(* IEC 61131-3 sources: programs/VI-54/VI-54_20171205/VI-54_20171205/Stations/Screen/LseClass170718/Class/AccessControlUSBDetection, 1 file *)

(* ---- AccessControlUSBDetection.st ---- *)
//"no usb stick is found" value

#define NO_USB 16#FFFF

(*!
<Class
	Name               = "AccessControlUSBDetection"
	Revision           = "1.1"
	RealtimeTask       = "false"
	CyclicTask         = "false"
	BackgroundTask     = "false"
	Sigmatek           = "false"
	OSInterface        = "false"
	HighPriority       = "false"
	Automatic          = "false"
	UpdateMode         = "Prescan"
	SharedCommandTable = "true"
	Objectsize         = "(570,240)"
	Comment            = "This class detects USB-activity.&#13;&#10;Override global-methods USBDeviceIN and USBDeviceOUT for user-defined action on usb-event&#13;&#10;">
	<Channels>
		<Client Name="cFileSys" Required="false" Internal="false" Comment="object channel to FileOp (don&apos;t connect!)"/>
		<Client Name="coAccessControl" Required="true" Internal="false" Comment="object channel - Connect to AccessControlMain object"/>
	</Channels>
	<RevDoku>
		<Owner Company="Sigmatek"/>
		<Dokumentation Revision="1.1" Date="2015-09-22" Company="Sigmatek" Description="Creation."/>
	</RevDoku>
	<Network Name="AccessControlUSBDetection">
		<!-- List of Components in this network -->
		<Components>
			<Object
				Name       = "_base"
				Class      = "_Global"
				Position   = "(218,120)"
				Visualized = "false">
				<Channels>
					<Server Name="Server0"/>
					<Client Name="Lse"/>
				</Channels>
			</Object>
		</Components>
		<Comments>
		</Comments>
		<!-- List of Connections in this network -->
		<Connections>
			<Connection Source="this.Server0" Destination="_base.Server0" Vertices="(690,210),(518,210),"/>
			<Connection Source="_base.Lse" Destination="this.Lse" Vertices="(218,210),(38,210),"/>
		</Connections>
		<!-- Headerfiles -->
		<Options>
		</Options>
	</Network>
</Class>
*)
#pragma using _Global

AccessControlUSBDetection : CLASS
: _Global
	TYPE
	  Letters :
	  (
	    _A,
	    _B,
	    _C,
	    _D,
	    _E,
	    _F,
	    _G,
	    _H,
	    _I,
	    _J,
	    _K,
	    _L,
	    _M,
	    _N,
	    _O,
	    _P,
	    _Q,
	    _R,
	    _S,
	    _T,
	    _U,
	    _V,
	    _W,
	    _X,
	    _Y,
	    _Z
	  )$UDINT;
	  T_SerNum : ARRAY [0..20] OF CHAR;
	END_TYPE
  //Servers:
  //Clients:
	cFileSys 	: CltChCmd__FileSys;
	coAccessControl 	: CltChCmd_AccessControlMain;
  //Variables:
		DriveList : ARRAY [0..25] OF CHAR;

		OldDriveList : ARRAY [0..25] OF CHAR;

		SerNumArray : ARRAY [0..25] OF T_SerNum;

  //Functions:

	FUNCTION VIRTUAL GLOBAL Init;

	FUNCTION VIRTUAL GLOBAL IF_WindowRun
		VAR_INPUT
			whoami 	: ^_WHOAMI;
			pic 	: ^void;
			event 	: ^_EVENT;
		END_VAR;
				//! <Function Comment="Will be called when a usb-stick is plugged in or out. It checks if a serial number of the usb-stick is available." Name="CheckSerNum"/>
	FUNCTION CheckSerNum
		VAR_INPUT
			INorOUT 	: DINT;			//! <Variable Comment="1..usb-stick is plugged in&#13;&#10;2..usb-stick is plugged out" Name="CheckSerNum.INorOUT"/>
		END_VAR;
				//! <Function Comment="Will be called when a usb-stick is plugged in." Name="USBDeviceIN"/>
	FUNCTION VIRTUAL GLOBAL USBDeviceIN
		VAR_INPUT
			pSerNum 	: ^void;			//! <Variable Comment="Pointer to the serial number of the usb-stick." Name="USBDeviceIN.pSerNum"/>
		END_VAR;
				//! <Function Comment="Will be called if a plugged in usb-stick is unplugged." Name="USBDeviceOUT"/>
	FUNCTION VIRTUAL GLOBAL USBDeviceOUT
		VAR_INPUT
			pSerNum 	: ^void;			//! <Variable Comment="Pointer to the serial number of the usb-stick." Name="USBDeviceOUT.pSerNum"/>
		END_VAR;
  //Tables:
	FUNCTION @STD
		VAR_OUTPUT
			ret_code	: CONFSTATES;
		END_VAR;
	FUNCTION GLOBAL TAB @CT_;
END_CLASS;

#pragma usingLtd _FileSys
#pragma usingLtd AccessControlMain

#include " lsl_st_syssernum.h"

FUNCTION VIRTUAL GLOBAL AccessControlUSBDetection::IF_WindowRun
	VAR_INPUT
		whoami 	: ^_WHOAMI;
		pic 	: ^void;
		event 	: ^_EVENT;
	END_VAR

  //call method from baseclass
  _Global::IF_WindowRun(whoami, pic, event);

  if event^.ftype <> _EVENT_NONE then
    //Check if there is some action on the usb-port
    if ( event^.ftype = _EVENT_LASALOS ) & ( event^.scancode = 8 )then

      //Check if usb stick was pluged or draged
      if event^.modifier = 1 | event^.modifier = 2 then

        cFileSys.GetDriveListShort(drivelist:= #DriveList$CHAR); //Get DriveList

        CheckSerNum(INorOUT:=event^.modifier); //check which device was plugged | unplugged

      end_if;
    end_if;
  end_if;

END_FUNCTION

FUNCTION VIRTUAL GLOBAL AccessControlUSBDetection::Init

  //call method from base class
  _Global::init();

  if _firstscan then
   _memset(#OldDriveList, 0, sizeof(OldDriveList));

  end_if;

END_FUNCTION

FUNCTION AccessControlUSBDetection::CheckSerNum
	VAR_INPUT
		INorOUT 	: DINT;
	END_VAR
  VAR
    counter : DINT;
    PISysSernum : ^LSL_ISYSSERNUM;
    Drive : USINT;
    pChar   : ^CHAR;
    retcode : DINT;
    Found : BOOL;
  END_VAR

  //search for all changed USb drives
  for counter := 0 to 25 do

    //if the drive is a UsbDevice, the device has changed since last UsbEvent and the device is plugged in
    if DriveList[counter] = 16#0B & DriveList[counter] <> OldDriveList[counter] & INorOUT = 1 then

      //check if serial number available and not zero
      if OS_CILGET("ISYSSERNUM", #pISysSernum) then
      else

         Drive := 'a' + to_usint(counter);
         _memset(#SerNumArray[counter], 0, sizeof(T_SerNum));
         retcode := ISYSSERNUM_SERNUMGETPLCDRIVE( Drive, #SerNumArray[counter], 20 );
         pChar := #SerNumArray[counter][0];
         Found := FALSE;
         while pChar^ <> 0 do
           if (pChar^ = ' ') | (pChar^ = '0') then
             pChar += sizeof(CHAR);
           else
             Found := TRUE;
             exit;
           end_if;
         end_while;
      end_if;

      if Found then

        USBDeviceIN(#SerNumArray[counter][0]); //call the user definable IN-Method

      end_if;

    //...if the device is unplugged
    elsif OldDriveList[counter] = 16#0B &  DriveList[counter] <> OldDriveList[counter] & INorOUT = 2 then

      USBDeviceOUT(#SerNumArray[counter][0]); //call the user definable OUT-Method
      _memset(#SerNumArray[counter], 0, sizeof(T_SerNum)); //clear SerNum

    end_if;

  end_for;

  //copy the actual DriveList
  _memcpy(#OldDriveList, #DriveList, sizeof(OldDriveList));

END_FUNCTION

FUNCTION VIRTUAL GLOBAL AccessControlUSBDetection::USBDeviceIN
	VAR_INPUT
		pSerNum 	: ^void;
	END_VAR
#pragma warning(default:73)

  coAccessControl.NewStick(pSerNum);

END_FUNCTION

FUNCTION VIRTUAL GLOBAL AccessControlUSBDetection::USBDeviceOUT
	VAR_INPUT
		pSerNum 	: ^void;
	END_VAR
#pragma warning(default:73)

  coAccessControl.StickRemoved(pSerNum);

END_FUNCTION
